PROGRAM MainTestPart
VAR
	//******************write data to file or read data from file**************************//
	m_FB_CSV_TextMode_ReadWrite1:FB_CSV_TextMode_ReadWrite;	
	m_bWrite: BOOL;
	m_writedata:ARRAY[0..19,0..9] OF LREAL;
	m_bRead:BOOL;
	m_readdata:ARRAY[0..10000,0..120] OF LREAL;
	
	
	
	
	//***************************single arm test related data****************************//
	m_armSelect:INT:=1;
	m_writeStart:BOOL;
	m_writeFinished:BOOL;
	m_writeStep:INT:=-1;
	m_fileId:INT;
	sFileName:T_MaxString;
	
	//data
	m_time:LREAL;
	m_row,m_col:INT;
	m_testDataWriteEnable:BOOL;	
	m_jntTrqD2,m_jntTrqD3:ARRAY[0..(gvl_const.g_writeDataNum-1),0..6] OF LREAL;
	m_jntPosD2,m_jntPosD3:ARRAY[0..(gvl_const.g_writeDataNum-1),0..6] OF LREAL;
	m_cmdDHjntPosD2,m_cmdDHjntPosD3:ARRAY[0..(gvl_const.g_writeDataNum-1),0..6] OF LREAL;
	m_data:ARRAY[0..(gvl_const.g_writeDataNum-1),0..6] OF LREAL;
	
	//pointer to global variables
	g_pcmdDHJntPosD2,g_pJntPosD2,g_pJntTrqD2:POINTER TO ARRAY[1..g_mArmNum,1..g_mJntNum,1..gvl_const.g_recordDataNum] OF LREAL;
	g_pcmdDHJntPosD3,g_pJntPosD3,g_pJntTrqD3:POINTER TO ARRAY[1..g_mArmNum,1..g_mJntNum,1..gvl_const.g_recordDataNum] OF LREAL;
	
	//data from global variables
	m_cmdDHJntPosD2_data,m_JntPosD2_data,m_JntTrqD2_data:ARRAY[1..g_mArmNum,1..g_mJntNum,1..gvl_const.g_recordDataNum] OF LREAL;
	m_cmdDHJntPosD3_data,m_JntPosD3_data,m_JntTrqD3_data:ARRAY[1..g_mArmNum,1..g_mJntNum,1..gvl_const.g_recordDataNum] OF LREAL;
	
	
	
	
	//**********************************write precision test data**********************************//
	m_armMatId:INT:=1;
	m_matWriteStep:INT:=-1;
	m_matrixData:ARRAY[0..3,0..3] OF LREAL;
	m_frontPose:ST_Frame;
	m_pfrontPose:POINTER TO ST_Frame;
	
	
	//*****************************Variables related to precision testing******************************//
	m_uiControlMode:ARRAY[1..2,0..GVL_Const.g_controlModeNum] OF BOOL;	
	m_uiControlModeL:ARRAY[1..2,0..GVL_Const.g_controlModeNum] OF BOOL;
	m_controlModeInit:ARRAY[1..2,0..GVL_Const.g_controlModeNum] OF BOOL;
    m_controlMode_TRIG:ARRAY[1..2,0..GVL_Const.g_controlModeNum] OF  R_TRIG;
	m_controlMode_FTRIG:ARRAY[1..2,0..GVL_Const.g_controlModeNum] OF  F_TRIG;	
	
	//unit function
	m_unitFun:FB_UnitTransform;
	
	//basic function
	m_basicFun:FB_BasicFun;
END_VAR

//write the data to file example
dataWriteExp();

//write the global data
writeArmTestData();

//HMI for accuracy test
HmiMid();
controlSignalAnalysis();

//write data related to precision test
writePrecisionData();

//information update
infoUpdate();

METHOD armInfoUpdate : BOOL
VAR_IN_OUT CONSTANT
	//i_slaveIdx :INT;
	//i_shoulderPose :ST_Frame;
	i_masterArm :FB_MasterArm;
	//i_slaveStatus :ST_SlaveStatus;
END_VAR
VAR
	i: INT;
	k:INT;
END_VAR

//update system information
FOR i:=1 TO g_mJntNum BY 1 DO
	k:=i_masterArm.armIdx;
	
	//motor input and output information
	g_systemInfo.m_armJntInfo[k,i].m_motorInput:=i_masterArm.m_joints[i].m_motorInputs;
	g_systemInfo.m_armJntInfo[k,i].m_motorOutput:=i_masterArm.m_joints[i].m_motorOutputs;
	
	//joint position and max/min
	g_systemInfo.m_armJntInfo[k,i].m_curJntPos:=i_masterArm.curJntPos[i];
	g_systemInfo.m_armJntInfo[k,i].m_jntMax:=GVL_ArmJointParameters.g_maxJntPos[k,i];
	g_systemInfo.m_armJntInfo[k,i].m_jntMin:=GVL_ArmJointParameters.g_minJntPos[k,i];
	
	//state machine
	g_systemInfo.m_masterArmState[k]:=MasterArmControl.m_masterRobot.m_masterArmState[k];
END_FOR



//update system information
FOR i:=1 TO g_mJntNum BY 1 DO
	k:=i_masterArm.armIdx;
	
	//motor input and output information
	g_systemInfo.m_armInfo[k].m_motorInput[i]:=i_masterArm.m_joints[i].m_motorInputs;
	g_systemInfo.m_armInfo[k].m_motorOutput[i]:=i_masterArm.m_joints[i].m_motorOutputs;
	
	//joint position and max/min	
	g_systemInfo.m_armJntInfo[k,i].m_jntMax:=GVL_ArmJointParameters.g_maxJntPos[k,i];
	g_systemInfo.m_armJntInfo[k,i].m_jntMin:=GVL_ArmJointParameters.g_minJntPos[k,i];
	
	//state machine
	g_systemInfo.m_masterArmState[k]:=MasterArmControl.m_masterRobot.m_masterArmState[k];
END_FOR

g_systemInfo.m_armInfo[k].m_curJntPos:=i_masterArm.curJntPos;
g_systemInfo.m_armInfo[k].m_curLinkPos:=i_masterArm.curLinkPos;
g_systemInfo.m_armInfo[k].m_curJntPosDegMM:=m_unitFun.masterArmUnit2User(i_dataSystem:= i_masterArm.curJntPos);
g_systemInfo.m_armInfo[k].m_curJntVelDegMM:=m_unitFun.masterArmUnit2User(i_dataSystem:= i_masterArm.curJntVel);
END_METHOD

METHOD carInfoUpdate : BOOL
VAR_INPUT
	m_masterCart :FB_MasterCart;
END_VAR

VAR
	i: INT;
END_VAR

//update system information
FOR i:=1 TO 4 BY 1 DO
	//motor input and output information
	g_systemInfo.m_cartJntInfo[i].m_motorInput:=m_masterCart.m_cartJoints[i].m_motorInputs;
	g_systemInfo.m_cartJntInfo[i].m_motorOutput:=m_masterCart.m_cartJoints[i].m_motorOutputs;
	
	//joint position and max/min
	g_systemInfo.m_cartJntInfo[i].m_curJntPos:=m_masterCart.m_curJntPos[i];
	g_systemInfo.m_cartJntInfo[i].m_jntMax:=GVL_CartJointParameters.g_maxJntPos[i];
	g_systemInfo.m_cartJntInfo[i].m_jntMin:=GVL_CartJointParameters.g_minJntPos[i];
END_FOR


//update system information
FOR i:=1 TO 4 BY 1 DO
	//motor input and output information
	g_systemInfo.m_cartInfo.m_motorInput[i]:=m_masterCart.m_cartJoints[i].m_motorInputs;
	g_systemInfo.m_cartInfo.m_motorOutput[i]:=m_masterCart.m_cartJoints[i].m_motorOutputs;		
END_FOR

//joint position and max/min
g_systemInfo.m_cartInfo.m_curJntPos:=m_masterCart.m_curJntPos;
g_systemInfo.m_cartInfo.m_curLinkPos:=m_masterCart.m_curLinkPos;
g_systemInfo.m_cartInfo.m_curJntPosDegMM:=m_unitFun.carArmUnit2User(i_dataSystem:= m_masterCart.m_curJntPos);
g_systemInfo.m_cartInfo.m_curJntVelDegMM:=m_unitFun.carArmUnit2User(i_dataSystem:= m_masterCart.m_curJntVel);


g_systemInfo.m_cartInfo.m_jntMax:=GVL_CartJointParameters.g_maxJntPos;
g_systemInfo.m_cartInfo.m_jntMin:=GVL_CartJointParameters.g_minJntPos;
END_METHOD

//*********Analyze the signals of the interactive interface*********//
METHOD controlSignalAnalysis : BOOL
VAR_INPUT
END_VAR

VAR
	i:INT;
	k:INT;
	activeJntPos,activeJntPosUser : vec7d;
	targetDHJntPos,targetDHJntPosUser:vec7d;
	m_armId:INT;
END_VAR
//go home signal
FOR m_armId:=1 TO g_mArmNum BY 1 DO
	FOR i:=1 TO g_mJntNum BY 1 DO
		IF (g_motionTest.m_goHome[m_armId][i]=TRUE) THEN
			g_motionTest.m_controlMode[m_armId]:=1;
			g_motionTest.m_startMotion[m_armId]:=TRUE;
			g_motionTest.m_jntPosIncMode[m_armId]:=FALSE;
			
			//give the target joint position
			FOR k:=1 TO g_mJntNum BY 1 DO
				targetDHJntPos[k]:=gvl_const.g_jntDHInitPos[m_armId,k];
			END_FOR
			targetDHJntPosUser:=m_unitFun.masterArmUnit2User(targetDHJntPos);
			
			g_motionTest.m_targetJntPos[m_armId]:=g_motionTest.m_armDHJntPos[m_armId];
			g_motionTest.m_targetJntPos[m_armId][i]:=targetDHJntPosUser[i];
			
			//exit for cycle
			EXIT;
		END_IF
	END_FOR
END_FOR



//go home signal---m_singleMotorStartMotion---m_singleMotorStartIncMotion
FOR m_armId:=1 TO g_mArmNum BY 1 DO
	FOR i:=1 TO g_mJntNum BY 1 DO
		IF (g_motionTest.m_goHome[m_armId][i]) OR (g_motionTest.m_singleMotorStartMotion[m_armId][i]) OR (g_motionTest.m_singleMotorStartIncMotion[m_armId][i]) THEN
			g_motionTest.m_controlMode[m_armId]:=1;
			g_motionTest.m_startMotion[m_armId]:=TRUE;				
			EXIT; //exit for cycle
		END_IF
	END_FOR
END_FOR



//cart joint go home---//监视器升降  监视器旋转  扶手升降  脚踏伸缩
FOR i:=1 TO 4 BY 1 DO
	IF (g_motionTest.m_goHomeCar[i]=TRUE) OR (g_motionTest.m_singleMotorStartMotion_Car[i]) OR (g_motionTest.m_singleMotorStartIncMotion_Car[i]) THEN
			g_motionTest.m_startMotionCar:=TRUE; //after motion finish,we should set the signal to false
			EXIT; //exit for cycle
	END_IF
END_FOR
END_METHOD

METHOD dataWriteExp : BOOL
VAR_INPUT
END_VAR

(*
m_FB_CSV_TextMode_ReadWrite1(	sNetId:= '', 	sFileName:='D:\file20241213.csv' , 	bBusy=> , 	bError=> , 	nErrorID=> , 	nErrorState=> );

m_FB_CSV_TextMode_ReadWrite1.M_WriteCsv(	bExecute:=m_bWrite , 	nMode:= FOPEN_MODEWRITE OR FOPEN_MODETEXT, 
	ptPointer:=ADR(m_writedata) , 	nRows:= 19, 	nColumns:=9 );

m_FB_CSV_TextMode_ReadWrite1.M_ReadCsv(bExecute:=m_bRead , ptPointer:= ADR(m_readdata), nRows:=10000 , nColumns:= 120);
IF NOT m_FB_CSV_TextMode_ReadWrite1.bBusy THEN
	m_bWrite:=FALSE;
	m_bRead:=FALSE;
END_IF
*)
END_METHOD

METHOD HmiMid : BOOL
VAR_INPUT
END_VAR
VAR
	i : INT;
	j : INT;
END_VAR
//data from ui
m_uiControlMode:=g_motionTest.m_uiArmMode;


//the interface relate to variable g_motionTest.m_uiArmMode
FOR i:=1 TO 2  DO
	FOR j:=1 TO GVL_Const.g_controlModeNum DO 
		//Monitoring button signal rising edge
		m_controlMode_TRIG[i,j](CLK:=m_uiControlMode[i,j],Q=>);
		
		IF (m_controlMode_TRIG[i,j].Q) AND (g_motionTest.m_controlMode[i]=0) THEN 			
			g_motionTest.m_controlMode[i]:=j;			
		END_IF
		
		//Monitoring button signal falling edge
		m_controlMode_FTRIG[i,j](CLK:=m_uiControlMode[i,j]);
	END_FOR	
	
	//If the accuracy test or workspace test is in progress, click the return to origin button to exit the accuracy test
	IF (g_motionTest.m_MSPrecisionTest[i]=TRUE) THEN
		IF (m_uiControlMode[i,6]=TRUE) THEN
			g_motionTest.m_controlMode[i]:=0;
			g_motionTest.m_MSPrecisionTest[i]:=FALSE;
		END_IF
	END_IF		
END_FOR


//Upload variables for displaying button colors
g_motionTest.m_uiArmModeL:=m_controlModeInit;
FOR i:=1 TO 2  DO
	g_motionTest.m_uiArmModeL[i,g_motionTest.m_controlMode[i]]:=TRUE;
END_FOR


//If the motion ends, set the relevant variables to false
FOR i:=1 TO 2  DO
	IF g_motionTest.m_controlMode[i]<>0 THEN
		g_motionTest.m_startMotion[i]:=TRUE;
	ELSE
		g_motionTest.m_startMotion[i]:=FALSE;
	END_IF
END_FOR
END_METHOD

METHOD infoUpdate : BOOL
VAR_INPUT
	
END_VAR

VAR
	i:INT;
END_VAR

//update the system information
FOR i:= 1 TO 2 BY 1 DO
	IF (MasterArmControl.m_robotInit=TRUE) THEN
		armInfoUpdate(i_masterArm:= MasterArmControl.m_masterRobot.m_masterArms[i]);
	END_IF	
END_FOR

//cart information
IF (CartControl.m_cartInit=TRUE) THEN
	carInfoUpdate(m_masterCart:= CartControl.m_masterCart);
END_IF
END_METHOD

METHOD writeArmTestData : BOOL
VAR_INPUT
END_VAR

VAR
	i,j:INT;
END_VAR

FOR i:=1 TO 2 BY 1 DO
	IF (g_frictionTest.m_writeData[i]=TRUE) THEN
		g_frictionTest.m_writeData[i]:=FALSE;
		m_armSelect:=i;
		m_writeStart:=TRUE;
	END_IF
END_FOR


IF (m_writeStart=TRUE) THEN
	m_writeStep:=0;
	m_writeStart:=FALSE;
	m_writeFinished:=FALSE;
END_IF


CASE m_writeStep OF
	0: //init parameters		
		m_row:=gvl_const.g_writeDataNum-1;
		m_col:=6;	
		
		g_pcmdDHJntPosD2:=ADR(g_frictionTest.m_cmdDHJntPosD2); g_pcmdDHJntPosD3:=ADR(g_frictionTest.m_cmdDHJntPosD3);
		g_pJntPosD2:=ADR(g_frictionTest.m_jntPosD2); g_pJntPosD3:=ADR(g_frictionTest.m_jntPosD3);
		g_pJntTrqD2:=ADR(g_frictionTest.m_jntTrqD2);  g_pJntTrqD3:=ADR(g_frictionTest.m_jntTrqD3);
		
		m_cmdDHJntPosD2_data:=g_pcmdDHJntPosD2^;	m_cmdDHJntPosD3_data:=g_pcmdDHJntPosD3^;
		m_JntPosD2_Data:=g_pJntPosD2^;	m_JntPosD3_Data:=g_pJntPosD3^;
		m_JntTrqD2_Data:=g_pJntTrqD2^;	m_JntTrqD3_Data:=g_pJntTrqD3^;
		
		FOR i:=0 TO m_col BY 1 DO
			FOR j:=0 TO m_row BY 1 DO
				m_cmdDHjntPosD2[j,i]:=m_cmdDHJntPosD2_data[m_armSelect,i+1,j+1]; m_cmdDHjntPosD3[j,i]:=m_cmdDHJntPosD3_data[m_armSelect,i+1,j+1];
				m_jntPosD2[j,i]:=m_JntPosD2_Data[m_armSelect,i+1,j+1]; m_jntPosD3[j,i]:=m_JntPosD3_Data[m_armSelect,i+1,j+1];
				m_jntTrqD2[j,i]:=m_JntTrqD2_Data[m_armSelect,i+1,j+1]; m_jntTrqD3[j,i]:=m_JntTrqD3_Data[m_armSelect,i+1,j+1];
			END_FOR
		END_FOR
				
		(*
		FOR i:=0 TO m_row BY 1 DO
			FOR j:=0 TO m_col BY 1 DO
				m_jntPosD2[i,j]:=i+1;
				m_jntTrqD2[i,j]:=i+1;
				m_jntPosD3[i,j]:=i+1;
				m_jntTrqD3[i,j]:=i+1;
			END_FOR
		END_FOR	
		*)
				
		m_fileId:=0;
		m_time:=0;
		m_writeStep:=10;
	
		
	10: //enable
		m_fileId:=m_fileId+1;
		IF (m_fileId=1) THEN
			sFileName:='C:\file1.txt';
			m_data:=m_jntPosD2;
		ELSIF (m_fileId=2) THEN
			sFileName:='C:\file2.txt';
			m_data:=m_jntPosD3;
		ELSIF (m_fileId=3) THEN
			sFileName:='C:\file3.txt';
			m_data:=m_jntTrqD2;
		ELSIF (m_fileId=4) THEN
			sFileName:='C:\file4.txt';
			m_data:=m_jntTrqD3;
		ELSIF (m_fileId=5) THEN
			sFileName:='C:\file5.txt';
			m_data:=m_cmdDHjntPosD2;
		ELSIF (m_fileId=6) THEN
			sFileName:='C:\file6.txt';
			m_data:=m_cmdDHjntPosD3;
		END_IF	
		m_testDataWriteEnable:=TRUE;
		m_writeStep:=20;
		
				
	20: //write the joint position
		m_FB_CSV_TextMode_ReadWrite1(	sNetId:= '', 	sFileName:=sFileName , 	bBusy=> , 	bError=> , 	nErrorID=> , 	nErrorState=> );
		m_FB_CSV_TextMode_ReadWrite1.M_WriteCsv(	bExecute:=m_testDataWriteEnable , 	nMode:= FOPEN_MODEWRITE OR FOPEN_MODETEXT, 
			ptPointer:=ADR(m_data) , 	nRows:= INT_TO_UINT(m_row), 	nColumns:=INT_TO_UINT(m_col) );
			
		//timer
		m_time:=m_time+0.010;
		
		IF (NOT m_FB_CSV_TextMode_ReadWrite1.bBusy) THEN
			m_FB_CSV_TextMode_ReadWrite1.M_WriteCsv(	bExecute:=FALSE , 	nMode:= FOPEN_MODEWRITE OR FOPEN_MODETEXT, 
			ptPointer:=ADR(m_data) , 	nRows:= INT_TO_UINT(m_row), 	nColumns:=INT_TO_UINT(m_col) );
			m_testDataWriteEnable:=FALSE;
			m_writeStep:=30;
			m_time:=0;
		END_IF
	
		
	30: //enable
		m_time:=m_time+0.010;
		IF (m_time>1) THEN
			m_time:=0;
			
			IF (m_fileId>=6) THEN
				m_writeStep:=40;
			ELSE
				m_testDataWriteEnable:=TRUE;
				m_writeStep:=10;
			END_IF			
		END_IF		
		

	40: //end
		m_writeFinished:=TRUE;
		m_writeStep:=-1;

		
	-1: //
END_CASE


//data write flag
i:=LIMIT(1,m_armSelect,2);
IF (m_writeStep=10) THEN	
	g_frictionTest.m_duringWriteData[i]:=TRUE;
ELSIF (m_writeStep=40) THEN
	g_frictionTest.m_duringWriteData[i]:=FALSE;
END_IF
END_METHOD

METHOD writePrecisionData : BOOL
VAR_INPUT
	
END_VAR
VAR
	i,j:INT;
END_VAR


FOR i:=1 TO 2 BY 1 DO
	IF (g_motionTest.m_writeData[i]=TRUE) THEN
		g_motionTest.m_writeData[i]:=FALSE;
		m_armMatId:=i;
		m_matWriteStep:=0;
	END_IF
END_FOR


CASE m_matWriteStep OF
	0: //prepare for the data
		m_pfrontPose:=ADR(g_motionTest.m_frontPose[m_armMatId]);
		m_frontPose:=m_pfrontPose^;
		
		//m_frontPose:=g_motionTest.m_frontPose[m_armMatId];
		FOR i:=1 TO 3 BY 1 DO			
			FOR j:=1 TO 3 BY 1 DO
				m_matrixData[i-1,j-1]:=m_frontPose.m_rot[i,j];
			END_FOR
		END_FOR
		
		FOR i:=1 TO 3 BY 1 DO
			m_matrixData[i-1,4-1]:=m_frontPose.m_pos[i];
		END_FOR
		m_matrixData[4-1,4-1]:=1;
		m_matWriteStep:=10;
		
		
	10:
		IF (m_armMatId=1) THEN
			sFileName:='C:\arm1.txt';
		ELSIF (m_armMatId=2) THEN
			sFileName:='C:\arm2.txt';
		END_IF
		
		m_row:=3;
		m_col:=3;
		m_time:=0;
		m_matWriteStep:=20;
		
		
	20: //write the joint position
		m_FB_CSV_TextMode_ReadWrite1(	sNetId:= '', 	sFileName:=sFileName , 	bBusy=> , 	bError=> , 	nErrorID=> , 	nErrorState=> );
		m_FB_CSV_TextMode_ReadWrite1.M_WriteCsv(	bExecute:=TRUE , 	nMode:= FOPEN_MODEWRITE OR FOPEN_MODETEXT, 
			ptPointer:=ADR(m_matrixData) , 	nRows:= INT_TO_UINT(m_row), 	nColumns:=INT_TO_UINT(m_col) );
			
		//timer
		m_time:=m_time+0.010;
		
		IF (NOT m_FB_CSV_TextMode_ReadWrite1.bBusy) THEN
			m_FB_CSV_TextMode_ReadWrite1.M_WriteCsv(	bExecute:=FALSE , 	nMode:= FOPEN_MODEWRITE OR FOPEN_MODETEXT, 
			ptPointer:=ADR(m_matrixData) , 	nRows:= INT_TO_UINT(m_row), 	nColumns:=INT_TO_UINT(m_col) );
			m_matWriteStep:=30;
			m_time:=0;
		END_IF
	
	
	30: //end
		m_matWriteStep:=-1;

		
	-1: //
END_CASE
END_METHOD

END_PROGRAM

(* stored: Version 1.1.0.1, ProductVersion 3.1.4024.11
   POU MainTestPart: Id {b83618ba-430f-4dc7-b8e8-725dcbac1ae2}, SpecialFunc None
   Method armInfoUpdate: Id {a7405eea-71fb-4e9b-be9b-5854851bcf65}
   Method carInfoUpdate: Id {88999e7e-7139-439c-aa60-34b95dafb49b}
   Method controlSignalAnalysis: Id {76d4e0aa-8494-4bf3-9bc8-a41cc2549c3d}
   Method dataWriteExp: Id {83e2b061-240b-48f5-a37e-40e2d8eb7275}
   Method HmiMid: Id {9a887a90-c99e-4390-abdb-ad0ecd202ca8}
   Method infoUpdate: Id {b5ebbaa2-522b-48df-8c3d-8db966613fb9}
   Method writeArmTestData: Id {75371ddd-c0a5-4294-8245-87433006a1e9}
   Method writePrecisionData: Id {029cd9d3-0755-4d4e-9858-76805cdd3ded} *)
